// TIA Portal V17 export
BLOCK "FB_Graph"   // ObjectSW20, GRAPH
BEGIN
// graph sequence
END_BLOCK
